# EPICS autosave request: iocBoot/ioc13ida_CD_Mono_XPS/auto_positions.req
file "CARS_motor_positions.req",         P=$(P), M=m57
file "CARS_motor_positions.req",         P=$(P), M=m58
file "CARS_motor_positions.req",         P=$(P), M=m59
file "CARS_motor_positions.req",         P=$(P), M=m60
file "CARS_motor_positions.req",         P=$(P), M=m61
